% RSLogix 500 project DIGITAL_ROTAMETER.RSS, saved by version 8.30.00.16 %
PROJECT "PROC1"    % processor: Bul.1763 MicroLogix 1100 Series B %

PROGRAM FILES
  LAD 2   9 rungs

DATA FILES
  O0 OUTPUT  4 elements
  I1 INPUT  6 elements
  S2 STATUS  66 elements
  B3 BINARY  1 elements
  T4 TIMER  3 elements
  C5 COUNTER  1 elements
  R6 CONTROL  1 elements
  N7 INTEGER  1 elements
  F8 FLOAT  2 elements

LADDER 2
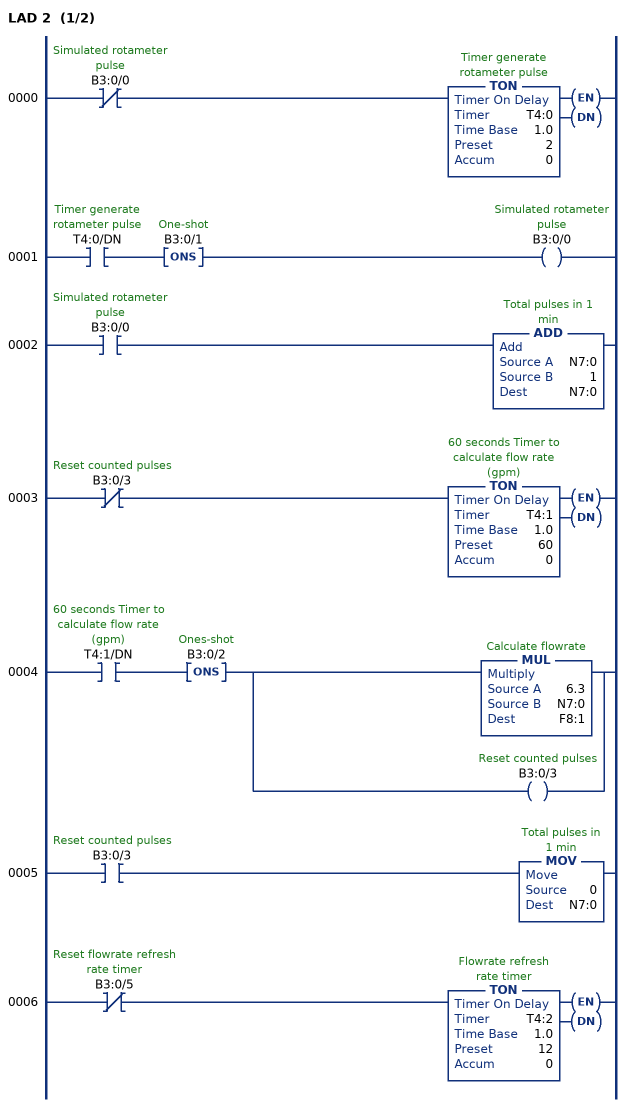
% Rung: 0 %
SOR XIO B3:0/0 TON T4:0 1.0 2 0 EOR
%   B3:0/0  "Simulated rotameter pulse" %
%   T4:0  "Timer generate rotameter pulse" %
% Rung: 1 %
SOR XIC T4:0/DN ONS B3:0/1 OTE B3:0/0 EOR
%   T4:0  "Timer generate rotameter pulse" %
%   B3:0/1  "One-shot" %
%   B3:0/0  "Simulated rotameter pulse" %
% Rung: 2 %
SOR XIC B3:0/0 ADD N7:0 1 N7:0 EOR
%   B3:0/0  "Simulated rotameter pulse" %
%   N7:0  "Total pulses in 1 min" %
% Rung: 3 %
SOR XIO B3:0/3 TON T4:1 1.0 60 0 EOR
%   B3:0/3  "Reset counted pulses" %
%   T4:1  "60 seconds Timer to calculate flow rate (gpm)" %
% Rung: 4 %
SOR XIC T4:1/DN ONS B3:0/2 BST MUL 6.3 N7:0 F8:1 NXB OTE B3:0/3 BND EOR
%   T4:1  "60 seconds Timer to calculate flow rate (gpm)" %
%   B3:0/2  "Ones-shot" %
%   N7:0  "Total pulses in 1 min" %
%   F8:1  "Calculate flowrate" %
%   B3:0/3  "Reset counted pulses" %
% Rung: 5 %
SOR XIC B3:0/3 MOV 0 N7:0 EOR
%   B3:0/3  "Reset counted pulses" %
%   N7:0  "Total pulses in 1 min" %
% Rung: 6 %
SOR XIO B3:0/5 TON T4:2 1.0 12 0 EOR
%   B3:0/5  "Reset flowrate refresh rate timer" %
%   T4:2  "Flowrate refresh rate timer" %

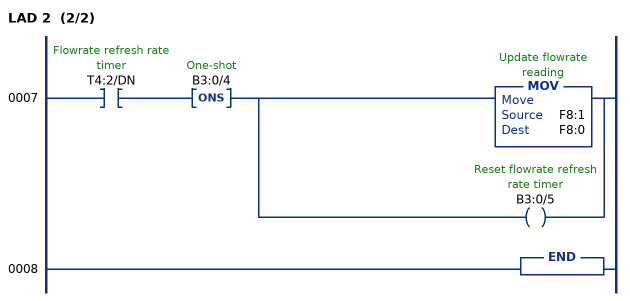
% Rung: 7 %
SOR XIC T4:2/DN ONS B3:0/4 BST MOV F8:1 F8:0 NXB OTE B3:0/5 BND EOR
%   T4:2  "Flowrate refresh rate timer" %
%   B3:0/4  "One-shot" %
%   F8:1  "Calculate flowrate" %
%   F8:0  "Update flowrate reading" %
%   B3:0/5  "Reset flowrate refresh rate timer" %
% Rung: 8 %
SOR END EOR

DATA TABLE (non-zero values as saved)
DATA T4
% .PRE .ACC %
% T4:0 % 2 0
% T4:1 % 60 0
% T4:2 % 12 0
